TYPE ST_Router_params :
STRUCT
	IP_TELTONIKA		: STRING(16) := '192.168.001.001';
	MBPort_TELTONIKA 	: UINT := 502;
	T_MBTimeout			: TIME := T#200MS;
	MinimumPhoneNumberLength	:	UINT := 10;
END_STRUCT
END_TYPE

(* stored: Version 1.1.0.1, ProductVersion 3.1.4024.12
   DUT ST_Router_params: Id {670cbed1-44dc-4e39-9f93-f60eade20940} *)
